(* PLC project  *)

CONFIGURATION Empty_Module_27
END_CONFIGURATION
